{attribute 'linkalways'}
{attribute 'no_explicit_call' := 'This FB is a CLASS and must be accessed using methods or properties'}
{attribute 'enable_dynamic_creation'}
FUNCTION_BLOCK Node_F_VN_FindReferenceKeyPointsInImageBRISKExp EXTENDS VisionNode
VAR
    ipSrcImage : _ITcVnImage;
    ipRefKeyPoints : _ITcVnContainer;
    ipRefDescriptors : _ITcVnImage;
    nRefImageWidth : _UDINT(0);
    nRefImageHeight : _UDINT(0);
    ipEdgePoints : _ITcVnContainer;
    fMaxDist : _REAL(-1.0);
    fMaxKnnRatio : _REAL(-1.0);
    eNormType : _ETcVnNormalizationType(ETcVnNormalizationType.TCVN_NT_HAMMING);
    ipSrcImageMask : _ITcVnImage;
    stBriskParams : _TcVnParamsBRISK;
    eAlgorithm : _ETcVnEstimationAlgorithm(ETcVnEstimationAlgorithm.TCVN_EA_RANSAC);
    fReprojThreshold : _LREAL(3.0);
    nMaxIterations : _UDINT(2000);
    fConfidence : _LREAL(0.995);
    hrPrev : _HRESULT(S_OK);
    aPerspectiveTransform : _TcVnMatrix3x3_LREAL;
    nNumberOfGoodMatches : _UDINT(0);
    nNumberOfInliers : _UDINT(0);
    hresult : _HRESULT(S_OK);
END_VAR

METHOD PUBLIC Clone : I_Node
VAR
    pNode : POINTER TO Node_F_VN_FindReferenceKeyPointsInImageBRISKExp;
END_VAR
pNode := __NEW(Node_F_VN_FindReferenceKeyPointsInImageBRISKExp);
Clone := pNode^;
END_METHOD

METHOD FB_init : BOOL
VAR_INPUT
    bInitRetains : BOOL;
    bInCopyCode : BOOL;
END_VAR
AddInput('ipSrcImage', ipSrcImage);
AddInput('ipRefKeyPoints', ipRefKeyPoints);
AddInput('ipRefDescriptors', ipRefDescriptors);
AddInput('nRefImageWidth', nRefImageWidth);
AddInput('nRefImageHeight', nRefImageHeight);
AddOutput('ipEdgePoints', ipEdgePoints);
AddParameter('fMaxDist', fMaxDist);
AddParameter('fMaxKnnRatio', fMaxKnnRatio);
AddParameter('eNormType', eNormType);
AddInput('ipSrcImageMask', ipSrcImageMask);
AddInput('stBriskParams', stBriskParams);
AddParameter('eAlgorithm', eAlgorithm);
AddParameter('fReprojThreshold', fReprojThreshold);
AddParameter('nMaxIterations', nMaxIterations);
AddParameter('fConfidence', fConfidence);
AddInput('hrPrev', hrPrev);
AddOutput('aPerspectiveTransform', aPerspectiveTransform);
AddOutput('nNumberOfGoodMatches', nNumberOfGoodMatches);
AddOutput('nNumberOfInliers', nNumberOfInliers);
AddOutput('hresult', hresult);
END_METHOD

METHOD PROTECTED OnExecute
VAR
    perspectiveTransform : TcVnMatrix3x3_LREAL;
    numberOfGoodMatches : UDINT;
    numberOfInliers : UDINT;
END_VAR
hresult.Value := F_VN_FindReferenceKeyPointsInImageBRISKExp(
    ipSrcImage := ipSrcImage.Value,
    ipRefKeyPoints := ipRefKeyPoints.Value,
    ipRefDescriptors := ipRefDescriptors.Value,
    nRefImageWidth := nRefImageWidth.Value,
    nRefImageHeight := nRefImageHeight.Value,
    ipEdgePoints := ipEdgePoints.Value,
    fMaxDist := fMaxDist.Value,
    fMaxKnnRatio := fMaxKnnRatio.Value,
    eNormType := eNormType.Value,
    ipSrcImageMask := ipSrcImageMask.Value,
    stBriskParams := stBriskParams.Value,
    eAlgorithm := eAlgorithm.Value,
    fReprojThreshold := fReprojThreshold.Value,
    nMaxIterations := nMaxIterations.Value,
    fConfidence := fConfidence.Value,
    hrPrev := hrPrev.Value,
    aPerspectiveTransform => perspectiveTransform,
    nNumberOfGoodMatches => numberOfGoodMatches,
    nNumberOfInliers => numberOfInliers);

aPerspectiveTransform.Value := perspectiveTransform;
nNumberOfGoodMatches.Value := numberOfGoodMatches;
nNumberOfInliers.Value := numberOfInliers;
END_METHOD

METHOD PUBLIC PreExecutionCheck
VAR_INPUT
    Check : I_PreExecutionChecks;
END_VAR
Check.IsTrue(ipSrcImage.IsValid, 'ipSrcImage must contain an image');
Check.IsTrue(ipSrcImage.HasChannelCount(1), 'ipSrcImage must have 1 channel');
IF ipSrcImageMask.Value <> 0 THEN
    Check.IsTrue(ipSrcImageMask.IsValid, 'ipSrcImageMask must contain an image when connected');
    Check.IsTrue(IsImage1SizeEqualToImage2Size(ipSrcImage.Value, ipSrcImageMask.Value), 'ipSrcImageMask must have the same size as ipSrcImage');
END_IF
Check.IsTrue(ipRefKeyPoints.IsValid, 'ipRefKeyPoints must contain a container');
Check.IsTrue(ipRefDescriptors.IsValid, 'ipRefDescriptors must contain an image');
Check.IsTrue(nRefImageWidth.Value > 0, 'nRefImageWidth must be greater than 0');
Check.IsTrue(nRefImageHeight.Value > 0, 'nRefImageHeight must be greater than 0');
Check.IsTrue((fMaxDist.Value = -1.0) OR (fMaxDist.Value >= 0.0), 'fMaxDist must be -1 to disable the filter, or at least 0');
Check.IsTrue((fMaxKnnRatio.Value = -1.0) OR
             ((fMaxKnnRatio.Value >= 0.0) AND (fMaxKnnRatio.Value <= 1.0)), 'fMaxKnnRatio must be -1 to disable the filter, or between 0 and 1');
Check.IsTrue((eNormType.Value = ETcVnNormalizationType.TCVN_NT_L1) OR
             (eNormType.Value = ETcVnNormalizationType.TCVN_NT_L2) OR
             (eNormType.Value = ETcVnNormalizationType.TCVN_NT_L2SQR) OR
             (eNormType.Value = ETcVnNormalizationType.TCVN_NT_HAMMING) OR
             (eNormType.Value = ETcVnNormalizationType.TCVN_NT_HAMMING2), 'Unsupported eNormType');
Check.IsTrue((eAlgorithm.Value = ETcVnEstimationAlgorithm.TCVN_EA_DEFAULT) OR
             (eAlgorithm.Value = ETcVnEstimationAlgorithm.TCVN_EA_LMEDS) OR
             (eAlgorithm.Value = ETcVnEstimationAlgorithm.TCVN_EA_RANSAC) OR
             (eAlgorithm.Value = ETcVnEstimationAlgorithm.TCVN_EA_RHO), 'Unsupported eAlgorithm');
// fReprojThreshold is only used by RANSAC and RHO.
Check.IsTrue(((eAlgorithm.Value <> ETcVnEstimationAlgorithm.TCVN_EA_RANSAC) AND
              (eAlgorithm.Value <> ETcVnEstimationAlgorithm.TCVN_EA_RHO)) OR
             (fReprojThreshold.Value > 0.0), 'fReprojThreshold must be greater than 0 for RANSAC and RHO');
Check.IsTrue(nMaxIterations.Value > 0, 'nMaxIterations must be greater than 0');
Check.IsTrue((fConfidence.Value > 0.0) AND (fConfidence.Value < 1.0), 'fConfidence must be between 0 and 1');
END_METHOD

END_FUNCTION_BLOCK

(* stored: Version 1.1.0.1, ProductVersion 3.1.4026.19
   POU Node_F_VN_FindReferenceKeyPointsInImageBRISKExp: Id {952f0c10-0a5c-4af9-8a40-4cc528b7a5d9}, SpecialFunc None
   Folder Constructor: Id {ae17d10e-1e71-4054-b0ab-ac9d23998933}
   Method Clone: Id {7196cf48-131d-41a2-ad94-03adc5c941af}
   Method FB_init: Id {e664dfdd-3580-42de-9298-a19f26b5a58f}
   Method OnExecute: Id {119dfad9-ad5d-4959-9774-b780435f7414}
   Method PreExecutionCheck: Id {d5c7e9a7-fbac-4e39-8eaa-7785242b7c8b} *)
